(* PLC project Tc2_Utilities.FB_ScopeServerControl Demo, tc3-libraries-kb TwinCAT 3.1 *)
(* stored: creationDateTime 2026-05-10T20:00:00, modificationDateTime 2026-05-10T20:00:00 *)

PROGRAM P_Demo_FB_ScopeServerControl
  VAR
    fbFB_ScopeServerControl : FB_ScopeServerControl;  (* Tc2_Utilities.FB_ScopeServerControl 实例 *)
    arg_sNetId : T_AmsNetId;  (* VAR_INPUT sNetId *)
    arg_eReqState : E_ScopeServerState;  (* VAR_INPUT eReqState *)
    arg_sConfigFile : STRING;  (* VAR_INPUT sConfigFile *)
    arg_sSaveFile : STRING;  (* VAR_INPUT sSaveFile *)
    arg_tTimeout : TIME;  (* VAR_INPUT tTimeout *)
    arg_bExternalTriggerEvent : BOOL;  (* VAR_INPUT bExternalTriggerEvent *)
    out_bBusy : BOOL;  (* VAR_OUTPUT bBusy *)
    out_bDone : BOOL;  (* VAR_OUTPUT bDone *)
    out_bError : BOOL;  (* VAR_OUTPUT bError *)
    out_nErrorId : UDINT;  (* VAR_OUTPUT nErrorId *)
  END_VAR

            // ============================================================
// Tc2_Utilities.FB_ScopeServerControl 演示程序（FB 实例）
// ============================================================
// 验证步骤：
//   1. 引用 Tc2_Utilities（及依赖类型所在库 Tc2_System 等）
//   2. 编译 + 登录
//   3. 按 doc.md 给 arg_* 赋值
//   4. 在线监视 out_* / io_* 输出
// ============================================================

fbFB_ScopeServerControl(
    sNetId := arg_sNetId,
    eReqState := arg_eReqState,
    sConfigFile := arg_sConfigFile,
    sSaveFile := arg_sSaveFile,
    tTimeout := arg_tTimeout,
    bExternalTriggerEvent := arg_bExternalTriggerEvent,
    bBusy => out_bBusy,
    bDone => out_bDone,
    bError => out_bError,
    nErrorId => out_nErrorId
);

          
END_PROGRAM
